// TIA Portal V18 export
FUNCTION "Alram_Scroll" : Void   // FC15, LAD
{ S7_Optimized_Access := 'TRUE' }
VERSION : 0.1
// stored: AutoNumber true, IsIECCheckEnabled false, SetENOAutomatically false, UDAEnableTagReadback false
   VAR CONSTANT
      "AlramDisplay time" : DInt := 2000;
   END_VAR
BEGIN

REGION Network 1
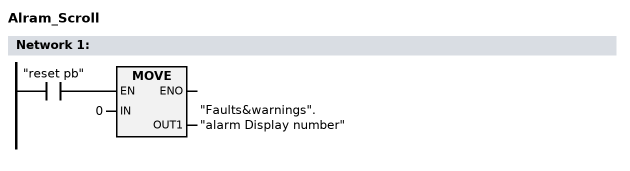
   RUNG wire#powerrail
      Contact( "reset pb" )
      Move(in := 0, out1 => "Faults&warnings"."alarm Display number")
   END_RUNG
   // the same network as SCL:
   IF "reset pb" THEN "Faults&warnings"."alarm Display number" := 0; END_IF;
END_REGION
END_FUNCTION
